PROGRAM MAIN
VAR PERSISTENT
	TubeSelection		: ARRAY[1..5] OF ST_TubeParameters; // array of tube parameters saved in memory
END_VAR
VAR
	CutOffValve	AT %Q*	: BOOL;
	Tube				: ST_TubeParameters;		// parameters in use by the machine
	TubeHmi				: ST_TubeParameters;		// parameters to edit in the hmi
	
	TubeIndicator		: ARRAY[1..5] OF BOOL := [TRUE, FALSE, FALSE, FALSE, FALSE];		// indicator as to which tube is in use
	
	fbSlitter			: FB_Slitter;				// object of machine
	Frame				: FB_Frame;	
	eCommand			: Tc3_PackML_V2.E_PMLCommand;
	eModeCommand		: DINT := E_PMLProtectedUnitMode.ePMLProtUnitMode_Production;
	eState				: Tc3_PackML_V2.E_PMLState;
	sState				: STRING;
	eMode				: DINT;

	TONhmi				: TON;
	TONidle				: TON := (PT := T#2M);
	ntStartProcess		: NT_StartProcess;

	bSave				: BOOL;
	bProcessing			: BOOL;
	bFailed				: BOOL;
	bPassed				: BOOL;
	fbWritePersistent	: FB_WritePersistentData;

	i					: INT;
	
	bOperation			: BOOL;
	bManual				: BOOL;
	bProductSettings	: BOOL;
	bMachineSettings	: BOOL;
	hmiStatus			: STRING := 'OK';
	PressureOn			: BOOL;
	PressureOnTon		: TON := (PT := T#10S);
	PressureOffTon		: TON := (PT := T#2s);
	hmiReset			: BOOL;
	bInspect			: BOOL;
	bNoDetect			: BOOL;
	InspectCommands		: ST_InspectCommands;
	
	currentUser: WSTRING;
	actualCurrentUser: WSTRING;
	debug1			: INT;
	debug2			: INT;
	nIndex			: INT;
	j				: INT;
	readTubeParameter	: ST_TubeParameters;
	emptyTubeParameter	: ST_TubeParameters;
	FilesLoaded		: BOOL;
	rTrigWriteFiles	: R_TRIG;
	nWriteFiles		: INT;
	fbXmlSrvRead	: FB_XmlSrvRead;
	fbXmlSrvWrite	: FB_XmlSrvWrite;
	fbMessage		: FB_TcMessage;
	x : INT;
END_VAR
VAR PERSISTENT	
	iBatch				: ULINT;
	iCounter			: ULINT;
	iCountFailed		: UINT;
	hmiBatch			: ULINT;
	CycleCounter		: LREAL;
END_VAR

CutOffValve := TRUE;

// set up the event logger message
IF NOT fbMessage.EqualsToEventEntryEx(stOther := TC_EVENTS.SlitterEvents.TubeParameterChange) THEN
	fbMessage.CreateEx(TC_EVENTS.SlitterEvents.TubeParameterChange, 0);
	fbMessage.ipArguments.Clear();
END_IF

// load the config parameters on start up
A_ReadTubeParameters();

// display the current user
IF currentUser <> VisuElems.CurrentFullUserName THEN
	currentUser := VisuElems.CurrentFullUserName;
END_IF

IF bOperation THEN				// when switching to the Operation page
	bOperation := FALSE;
	FOR i:=1 TO 5 DO
		TubeIndicator[i] := FALSE;
	END_FOR
	TubeIndicator[1] := TRUE;
	Tube := TubeSelection[1];	// set the tube selection to the first tube on entering page
	TubeHmi := Tube;			// write the parameters to the HMI display
END_IF

IF bManual THEN
	bManual := FALSE;
	TubeHmi := Tube;	// write the parameters to the HMI display
						// do not change the selected tube
END_IF

IF bProductSettings THEN
	bProductSettings := FALSE;
	FOR i:=1 TO 5 DO
		TubeIndicator[i] := FALSE;
	END_FOR
	TubeIndicator[1] := TRUE;
	Tube := TubeSelection[1];	// on entering product page select the first tube
	TubeHmi := Tube;			// write the parameters to the HMI display
END_IF

IF bMachineSettings THEN
	bMachineSettings := FALSE;
	TubeHmi := Tube;
END_IF

//A_StartVisualization();
A_PackMlCommands();

// this must be called before the fbSlitter execution
// determines the tube that is selected 
FOR i := 1 TO 5 DO
	IF TubeIndicator[i] THEN
		Tube := TubeSelection[i];
	END_IF
END_FOR

// machine object
fbSlitter(
	eCommand := eCommand,
	eModeCommand := eModeCommand,
	Batch := hmiBatch,
	Tube := Tube,
	TubeHmi := TubeHmi,	// used only for manual commands
	Inspect := bInspect,
	InspectCmd := InspectCommands,
	CounterOut => iCounter,
	CountFailedOut => iCountFailed,
	BatchOut => iBatch,
	eState => eState,
	sState => sState,
	eMode => eMode);

IF eState <> E_PMLState.ePMLState_Undefined THEN
	A_MonitorParameters();
	A_WriteParameters();
END_IF	
A_StatusIndicator();
(*		
FOR i := 1 TO 5 DO
	IF TubeIndicator[i] THEN
		debug2 := debug2 + 1;		
		IF MEMCMP(ADR(Tube), ADR(TubeSelection[i]), SIZEOF(tube)) <> 0 THEN
			TubeHmi := Tube;		
			bSave := TRUE;
			debug1 := debug1 + 1;
		END_IF 
	END_IF
END_FOR
*)

ACTION A_MonitorParameters:
IF MEMCMP(ADR(TubeHmi), ADR(TubeSelection[i]), SIZEOF(TubeHmi)) <> 0 THEN
	IF TubeHmi.AdjustmentLength <> TubeSelection[i].AdjustmentLength THEN
		// Tube {0} Parameter {1} changed from {2} to {3}
		fbMessage.ipArguments.Clear();
		fbMessage.ipArguments.AddInt(i).AddString('AdjustmentLength');
		fbMessage.ipArguments.AddLReal(TubeSelection[i].AdjustmentLength).AddLReal(TubeHmi.AdjustmentLength);
		fbMessage.Send(0);
	END_IF
	IF TubeHmi.AdjustmentX <> TubeSelection[i].AdjustmentX THEN
		fbMessage.ipArguments.Clear();
		fbMessage.ipArguments.AddInt(i).AddString('AdjustmentX');
		fbMessage.ipArguments.AddLReal(TubeSelection[i].AdjustmentX).AddLReal(TubeHmi.AdjustmentX);
		fbMessage.Send(0);				
	END_IF
	IF TubeHmi.AdjustmentY <> TubeSelection[i].AdjustmentY THEN
		fbMessage.ipArguments.Clear();
		fbMessage.ipArguments.AddInt(i).AddString('AdjustmentY');
		fbMessage.ipArguments.AddLReal(TubeSelection[i].AdjustmentY).AddLReal(TubeHmi.AdjustmentY);
		fbMessage.Send(0);								
	END_IF
	IF TubeHmi.CutPositionX <> TubeSelection[i].CutPositionX THEN
		fbMessage.ipArguments.Clear();
		fbMessage.ipArguments.AddInt(i).AddString('CutPositionX');
		fbMessage.ipArguments.AddLReal(TubeSelection[i].CutPositionX).AddLReal(TubeHmi.CutPositionX);
		fbMessage.Send(0);												
	END_IF
	IF TubeHmi.CutPositionY <> TubeSelection[i].CutPositionY THEN
		fbMessage.ipArguments.Clear();
		fbMessage.ipArguments.AddInt(i).AddString('CutPositionY');
		fbMessage.ipArguments.AddLReal(TubeSelection[i].CutPositionY).AddLReal(TubeHmi.CutPositionY);
		fbMessage.Send(0);																
	END_IF
	IF TubeHmi.DepthOfPocket <> TubeSelection[i].DepthOfPocket THEN
		fbMessage.ipArguments.Clear();
		fbMessage.ipArguments.AddInt(i).AddString('DepthOfPocket');
		fbMessage.ipArguments.AddLReal(TubeSelection[i].DepthOfPocket).AddLReal(TubeHmi.DepthOfPocket);
		fbMessage.Send(0);																				
	END_IF
	IF TubeHmi.Description <> TubeSelection[i].Description THEN
		fbMessage.ipArguments.Clear();
		fbMessage.ipArguments.AddInt(i).AddString('Description');
		fbMessage.ipArguments.AddString(TubeSelection[i].Description).AddStringByValue(TubeHmi.Description);
		fbMessage.Send(0);																								
	END_IF
	IF TubeHmi.Diameter <> TubeSelection[i].Diameter THEN
		fbMessage.ipArguments.Clear();
		fbMessage.ipArguments.AddInt(i).AddString('Diameter');
		fbMessage.ipArguments.AddLReal(TubeSelection[i].Diameter).AddLReal(TubeHmi.Diameter);
		fbMessage.Send(0);																												
	END_IF
	IF TubeHmi.EjectPositionX <> TubeSelection[i].EjectPositionX THEN
		fbMessage.ipArguments.Clear();
		fbMessage.ipArguments.AddInt(i).AddString('EjectPositionX');
		fbMessage.ipArguments.AddLReal(TubeSelection[i].EjectPositionX).AddLReal(TubeHmi.EjectPositionX);
		fbMessage.Send(0);																												
	END_IF	
	IF TubeHmi.EjectPositionY <> TubeSelection[i].EjectPositionY THEN
		fbMessage.ipArguments.Clear();
		fbMessage.ipArguments.AddInt(i).AddString('EjectPositionY');
		fbMessage.ipArguments.AddLReal(TubeSelection[i].EjectPositionY).AddLReal(TubeHmi.EjectPositionY);
		fbMessage.Send(0);																												
	END_IF
	IF TubeHmi.InspectPositionX <> TubeSelection[i].InspectPositionX THEN
		fbMessage.ipArguments.Clear();
		fbMessage.ipArguments.AddInt(i).AddString('InspectPositionX');
		fbMessage.ipArguments.AddLReal(TubeSelection[i].InspectPositionX).AddLReal(TubeHmi.InspectPositionX);
		fbMessage.Send(0);																																
	END_IF
	IF TubeHmi.InspectPositionY <> TubeSelection[i].InspectPositionY THEN
		fbMessage.ipArguments.Clear();
		fbMessage.ipArguments.AddInt(i).AddString('InspectPositionY');
		fbMessage.ipArguments.AddLReal(TubeSelection[i].InspectPositionY).AddLReal(TubeHmi.InspectPositionY);
		fbMessage.Send(0);																																				
	END_IF
	IF TubeHmi.MaxHeight <> TubeSelection[i].MaxHeight THEN
		fbMessage.ipArguments.Clear();
		fbMessage.ipArguments.AddInt(i).AddString('MaxHeight');
		fbMessage.ipArguments.AddLReal(TubeSelection[i].MaxHeight).AddLReal(TubeHmi.MaxHeight);
		fbMessage.Send(0);																																								
	END_IF
	IF TubeHmi.MaxLength <> TubeSelection[i].MaxLength THEN
		fbMessage.ipArguments.Clear();
		fbMessage.ipArguments.AddInt(i).AddString('MaxLength');
		fbMessage.ipArguments.AddLReal(TubeSelection[i].MaxLength).AddLReal(TubeHmi.MaxLength);
		fbMessage.Send(0);																																												
	END_IF
	IF TubeHmi.MinHeight <> TubeSelection[i].MinHeight THEN
		fbMessage.ipArguments.Clear();
		fbMessage.ipArguments.AddInt(i).AddString('MinHeight');
		fbMessage.ipArguments.AddLReal(TubeSelection[i].MinHeight).AddLReal(TubeHmi.MinHeight);
		fbMessage.Send(0);																																																
	END_IF
	IF TubeHmi.MinLength <> TubeSelection[i].MinLength THEN
		fbMessage.ipArguments.Clear();
		fbMessage.ipArguments.AddInt(i).AddString('MinLength');
		fbMessage.ipArguments.AddLReal(TubeSelection[i].MinLength).AddLReal(TubeHmi.MinLength);
		fbMessage.Send(0);																																																				
	END_IF
	IF TubeHmi.ProductName <> TubeSelection[i].ProductName THEN
		fbMessage.ipArguments.Clear();
		fbMessage.ipArguments.AddInt(i).AddString('ProductName');
		fbMessage.ipArguments.AddString(TubeSelection[i].ProductName).AddString(TubeHmi.ProductName);
		fbMessage.Send(0);																																																				
	END_IF
	IF TubeHmi.ResultToleranceX <> TubeSelection[i].ResultToleranceX THEN
		fbMessage.ipArguments.Clear();
		fbMessage.ipArguments.AddInt(i).AddString('ResultToleranceX');
		fbMessage.ipArguments.AddLReal(TubeSelection[i].ResultToleranceX).AddLReal(TubeHmi.ResultToleranceX);
		fbMessage.Send(0);																																																				
	END_IF
	IF TubeHmi.ResultToleranceY <> TubeSelection[i].ResultToleranceY THEN
		fbMessage.ipArguments.Clear();
		fbMessage.ipArguments.AddInt(i).AddString('ResultToleranceY');
		fbMessage.ipArguments.AddLReal(TubeSelection[i].ResultToleranceY).AddLReal(TubeHmi.ResultToleranceY);
		fbMessage.Send(0);																																																								
	END_IF
	IF TubeHmi.VacuumThreshold <> TubeSelection[i].VacuumThreshold THEN
		fbMessage.ipArguments.Clear();
		fbMessage.ipArguments.AddInt(i).AddString('VacuumThreshold');
		fbMessage.ipArguments.AddLReal(TubeSelection[i].VacuumThreshold).AddLReal(TubeHmi.VacuumThreshold);
		fbMessage.Send(0);																																																								
	END_IF
END_IF
END_ACTION

ACTION A_PackMlCommands:
PressureOffTon(IN := frame.Pressure < 80);
IF PressureOffTon.Q THEN
	PressureOn := FALSE;
END_IF
PressureOnTON(IN := frame.Pressure > 80);
IF PressureOnTON.Q THEN
	PressureOn := TRUE;
END_IF

// pack ml commands
IF (NOT PressureOn OR hmiReset) AND FilesLoaded THEN
 	eCommand := E_PMLCommand.ePMLCommand_Abort;
	hmiReset := FALSE;
	IF NOT PressureOn THEN
		hmiStatus := 'Pressure<80PSIG';
	END_IF
ELSIF eMode = E_PMLProtectedUnitMode.ePMLProtUnitMode_Manual THEN
	hmiStatus := 'Manual Mode';
	IF eModeCommand = E_PMLProtectedUnitMode.ePMLProtUnitMode_Production THEN
		eCommand := E_PMLCommand.ePMLCommand_Abort;
		Frame.GreenLight := FALSE;
	ELSE
		CASE eState OF
			E_PMLState.ePMLState_Undefined: eCommand := E_PMLCommand.ePMLCommand_Abort;
			E_PMLState.ePMLState_Aborted: eCommand := E_PMLCommand.ePMLCommand_Clear;
			E_PMLState.ePMLState_Idle: eCommand := E_PMLCommand.ePMLCommand_Start;
			E_PMLState.ePMLState_Stopped: eCommand := E_PMLCommand.ePMLCommand_Reset;
			E_PMLState.ePMLState_Aborting: eCommand := E_PMLCommand.ePMLCommand_Undefined;
		END_CASE
	END_IF
ELSIF eMode = E_PMLProtectedUnitMode.ePMLProtUnitMode_Production THEN
	hmiStatus := 'Automatic Mode';
	IF eModeCommand = E_PMLProtectedUnitMode.ePMLProtUnitMode_Manual THEN
		eCommand := E_PMLCommand.ePMLCommand_Abort;
	ELSE
		CASE eState OF
			E_PMLState.ePMLState_Undefined:
				IF FilesLoaded THEN
					eCommand := E_PMLCommand.ePMLCommand_Abort;
				END_IF
			E_PMLState.ePMLState_Aborted:  
				//IF NOT Frame.Door1 AND NOT Frame.Door2 THEN
					eCommand := E_PMLCommand.ePMLCommand_Clear;
				//END_IF
			E_PMLState.ePMLState_Idle:
					Frame.GreenLight := Frame.Door1 AND Frame.Door2 AND Frame.Door3 AND Frame.Door4;
					IF Frame.GreenLight THEN
						hmiStatus := 'Ready';
					ELSE
						hmiStatus := 'Door Open';
					END_IF
					IF (Frame.ControlLeft AND Frame.ControlRight) AND Frame.GreenLight THEN
						eCommand := E_PMLCommand.ePMLCommand_Start;
						Frame.GreenLight := FALSE;
					END_IF
			E_PMLState.ePMLState_Complete: eCommand := E_PMLCommand.ePMLCommand_Reset;
														
			E_PMLState.ePMLState_Stopped: eCommand := E_PMLCommand.ePMLCommand_Reset;
			E_PMLState.ePMLState_Aborting: eCommand := E_PMLCommand.ePMLCommand_Undefined;			
		END_CASE
	END_IF
END_IF
END_ACTION

ACTION A_ReadTubeParameters:
x := x + 1;

CASE nIndex OF
	0: // read the info from the config file for the camera
		j := 1;
		nIndex := 10;
	10: // 
		fbXmlSrvRead.sXPath := CONCAT('/Configuration/TubeParameters/Tube', INT_TO_STRING(j));
		fbXmlSrvRead.pSymAddr := ADR(readTubeParameter);
		fbXmlSrvRead.cbSymSize := SIZEOF(readTubeParameter);
		fbXmlSrvRead.bExecute := TRUE;
		nIndex := 20;
	20: // wait for the info to load
		IF NOT fbXmlSrvRead.bBusy THEN
			fbXmlSrvRead.bExecute := FALSE;
			MEMCPY(ADR(TubeSelection[j]), ADR(readTubeParameter), SIZEOF(readTubeParameter));
			MEMCPY(ADR(readTubeParameter), ADR(emptyTubeParameter), SIZEOF(emptyTubeParameter));
			nIndex := 30;
			IF j >= 5 THEN
				nIndex := 30;
			ELSE
				nIndex := 10;
				j := j + 1;
			END_IF
		END_IF
	30: // set variables
		Tube := TubeSelection[1];
		TubeHmi := TubeSelection[1];
		TubeIndicator[1] := TRUE;
		bProcessing := FALSE;
		bPassed := FALSE;
		bFailed := FALSE;
		bNoDetect := FALSE;
		nIndex := 40;
	40: // wait here for files loaded
		IF fbSlitter.ReadParameters(Execute := TRUE) THEN
			fbSlitter.ReadParameters(Execute := FALSE);
			FilesLoaded := TRUE;
			nIndex := 50;
		END_IF
	50: // 
		
END_CASE

fbXmlSrvRead(
	sNetId:= '', 
	ePath:= E_OpenPath.PATH_GENERIC, 
	nMode:= XMLSRV_SKIPMISSING, 
	sFilePath:= 'C:\Configuration.xml');
END_ACTION

ACTION A_StartVisualization:
// start the hmi

TONhmi(IN := TRUE, PT := T#4S);
IF TONhmi.Q THEN
	ntStartProcess(
		NETID := '',
		PATHSTR := 'C:\TwinCAT\3.1\Components\Plc\Tc3PlcHmi\Tc3PlcHmi.exe',
		DIRNAME := 'C:\TwinCAT\3.1\Components\Plc\Tc3PlcHmi\',
		COMNDLINE := 'Tc3PlcHmi.exe',
		START := TRUE);
END_IF
END_ACTION

ACTION A_StatusIndicator:
// status indicator

IF eMode = E_PMLProtectedUnitMode.ePMLProtUnitMode_Production THEN
	CASE fbSlitter.Status OF
		0: // idle if idle is on for more than 2 minutes, remove the result
			TONidle(IN := TRUE);
			bProcessing := FALSE;
			IF TONidle.Q THEN
				bFailed := FALSE;
				bPassed := FALSE;	
				bNoDetect := FALSE;		
			END_IF
		1: // processing
			bProcessing := TRUE;
			bFailed := FALSE;
			bPassed := FALSE;
			bNoDetect := FALSE;
			TONidle(IN := FALSE);
		2: // pass
			bPassed := TRUE;
			bFailed := FALSE;
			bProcessing := FALSE;
			bNoDetect := FALSE;
		3: // fail	
			bPassed := FALSE;
			bFailed := TRUE;
			bProcessing := FALSE;
			bNoDetect := FALSE;
		4: // failed to detect
			bPassed := FALSE;
			bFailed := FALSE;
			bProcessing := FALSE;
			bNoDetect := TRUE;		
	END_CASE
ELSE
	bPassed := FALSE;
	bFailed := FALSE;
	bProcessing := FALSE;
END_IF
END_ACTION

ACTION A_WriteParameters:
// write persistent data 
rTrigWriteFiles(CLK := bSave);
IF rTrigWriteFiles.Q THEN
	fbSlitter.SaveParameters(Execute := FALSE);
	nWriteFiles := 10;
END_IF

IF NOT bSave THEN
	nWriteFiles := 0;
END_IF

CASE nWriteFiles OF
	10: // get the tube into memory
		FOR i := 1 TO 5 DO
			IF TubeIndicator[i] THEN
				A_MonitorParameters();
				TubeSelection[i] := TubeHmi;
				TubeSelection[i].Index := i;
			END_IF
		END_FOR
		j := 1;
		nWriteFiles := 20;
	20: // write the tube parameters
		MEMCPY(ADR(readTubeParameter), ADR(TubeSelection[j]), SIZEOF(readTubeParameter));
		fbXmlSrvWrite.bExecute := TRUE;
		fbXmlSrvWrite.cbSymSize := SIZEOF(readTubeParameter);
		fbXmlSrvWrite.pSymAddr := ADR(readTubeParameter);
		fbXmlSrvWrite.sXPath := CONCAT('/Configuration/TubeParameters/Tube', INT_TO_STRING(j));
		nWriteFiles := 30;
	30: // wait to complete
		IF NOT fbXmlSrvWrite.bBusy THEN
			fbXmlSrvWrite.bExecute := FALSE;
			IF j >= 5 THEN
				nWriteFiles := 40;
			ELSE
				j := j + 1;
				nWriteFiles := 20;
			END_IF
		END_IF
	40: // command slitter to save parameters
		IF fbSlitter.SaveParameters(Execute := TRUE) THEN
			fbSlitter.SaveParameters(Execute := FALSE);
			nWriteFiles := 50;
		END_IF
	50: // done state
		bSave := FALSE;
END_CASE

fbXmlSrvWrite(
	sNetId:= '', 
	ePath:= E_OpenPath.PATH_GENERIC, 
	nMode:= XMLSRV_SKIPMISSING, 
	sFilePath:= 'C:\Configuration.xml');
END_ACTION

END_PROGRAM

(* stored: Version 1.1.0.1, ProductVersion 3.1.4024.9
   POU MAIN: Id {8f3c7fd0-6d9b-4406-902d-14a13902ae94}, SpecialFunc None
   Action A_MonitorParameters: Id {11b27928-fe1e-4d76-9e99-f24f8c688575}
   Action A_PackMlCommands: Id {7dff5ef5-514a-4270-badc-d4173046ca34}
   Action A_ReadTubeParameters: Id {08beef19-af36-40fc-994a-42f92c970fef}
   Action A_StartVisualization: Id {28a6a13c-0164-45f7-82c3-d3ce337639c7}
   Action A_StatusIndicator: Id {fa378544-fe8e-49fa-b056-a4700d79bbe0}
   Action A_WriteParameters: Id {09528414-ba2a-4def-9a55-fdd92ee4ec57} *)
